(* PLC project Counter (OSIE), Unknown Unnamed 1 *)
(* stored: creationDateTime 2021-05-14T14:33:11, modificationDateTime 2021-05-17T11:58:28 *)

FUNCTION_BLOCK CounterST
  VAR_INPUT
    Reset : BOOL;
  END_VAR
  VAR_OUTPUT
    Out : INT;
  END_VAR
  VAR
    Cnt : INT;
  END_VAR
  VAR_EXTERNAL
    ResetCounterValue : INT;
  END_VAR

            IF Reset THEN
  Cnt := ResetCounterValue;
ELSE
  Cnt := Cnt + 1;
END_IF;

Out := Cnt;
          
END_FUNCTION_BLOCK

PROGRAM plc_prg
  VAR_INPUT
    Reset : BOOL;
  END_VAR
  VAR_OUTPUT
    Cnt0 : INT;
    Cnt1 : INT;
    Cnt2 : INT;
    Cnt3 : INT;
    Cnt4 : INT;
  END_VAR
  VAR
    CounterST0 : CounterST;
  END_VAR

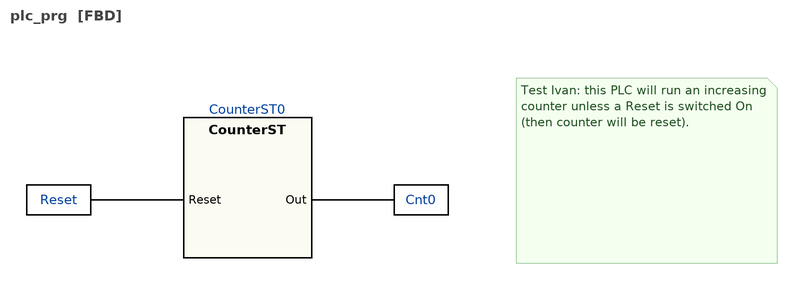
(* FBD diagram, written out as Structured Text *)
(* Test Ivan: this PLC will run an increasing counter unless a Reset is switched On (then counter will be reset). *)
CounterST0(Reset := Reset);
Cnt0 := CounterST0.Out;
END_PROGRAM

CONFIGURATION config
  VAR_GLOBAL
    ResetCounterValue : INT := 1000;
  END_VAR
  RESOURCE resource1 ON PLC
    TASK task0(INTERVAL := T#20ms, PRIORITY := 0);
    PROGRAM instance0 WITH task0 : plc_prg;
  END_RESOURCE
END_CONFIGURATION
